(* CODESYS project DrugiiiiiZadatak (1).project
   CustomField04_name: CustomField04
   CustomField06_name: CustomField06
   CustomField07_name: CustomField07
   CustomField09_name: CustomField09
   CustomField08_name: CustomField08
   CustomField02_name: CustomField02
   CustomField10_name: CustomField10
   CustomField01_name: CustomField01
   CustomField03_name: CustomField03
   CustomField05_name: CustomField05

Project tree, tasks and I/O mapping:
  MyController : TM238LFDC24DT, Schneider Electric, order no. TM238LFDC24DT, version 2.0.31.8
    application Application
      task MAST (cyclic, interval 20 ms, priority 15, watchdog 100 ms x 1) calls POU
      function HiddenPOU [ST]
      global variables GVL
      program POU [LD]
    CAN
    Embedded Functions
      HSC : HSC, Schneider Electric, version 2.0.31.8
        HSC
      PTO_PWM : PTO_PWM, Schneider Electric, version 2.0.31.8
        PTO_PWM
      IO : IO, Schneider Electric, version 2.0.31.8
          input  Application.POU.Tipkalo2 : BOOL  // IW0.I9
          input  Application.POU.Tipkalo1 : BOOL  // IW0.I10
          output Application.POU.Zelena1 : BOOL  // QW0.Q4
          output Application.POU.Zuta1 : BOOL  // QW0.Q5
          output Application.POU.Crvena1 : BOOL  // QW0.Q6
          unmapped channels: IW0, QW0
    Serial Line 1
      Modbus_Manager : Modbus_Manager, Schneider Electric, version 2.0.1.12
    Serial Line 2
      SoMachine_Network_Manager : SoMachine-Network_Manager, Schneider Electric, version 2.0.1.10
  MachineLayoutPicture
*)

// MyController/Application/GVL
VAR_GLOBAL
END_VAR

// MyController/Application/POU
PROGRAM POU
VAR
	Tipkalo1: BOOL;
	Tipkalo2: BOOL;
	brojilo: CTUD := (CV := 5, RESET := FALSE, PV := 0, LOAD := FALSE, CD := FALSE, CU := FALSE, QD := FALSE, QU := FALSE);
	Zelena1: BOOL;
	Crvena1: BOOL;
	Zuta1: BOOL;
	
	
	titraj1: TP := (Q := TRUE, PT := TIME#5000ms, ET := TIME#5000ms, IN := TRUE);
	pomocni: TP := (Q := TRUE, PT := TIME#400MS, ET := TIME#400MS, IN := FALSE);
	pomocni1: TON := (Q := FALSE, PT := TIME#400ms, ET := TIME#0ms, IN := FALSE);
	pomocni3: TON := (Q := TRUE, PT := TIME#400MS, ET := TIME#0MS, IN := TRUE);
END_VAR

VAR_OUTPUT
	
END_VAR

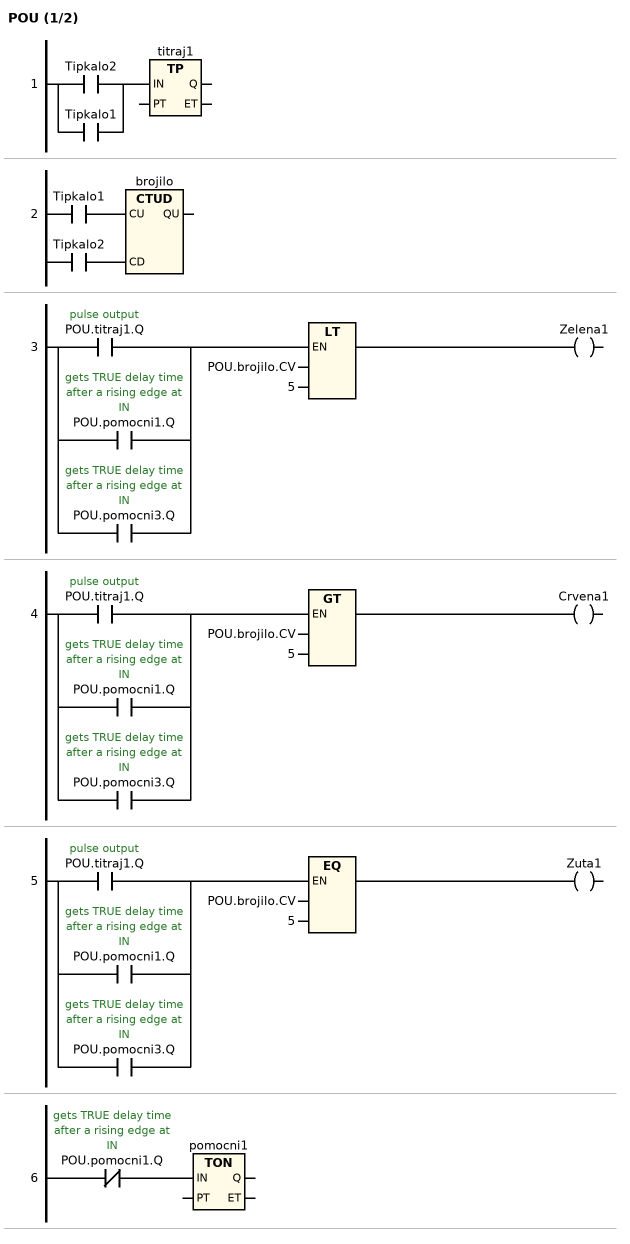
// NETWORK 1
titraj1(IN := Tipkalo2 OR Tipkalo1); // TP

// NETWORK 2
brojilo(CU := Tipkalo1, CD := Tipkalo2); // CTUD

// NETWORK 3
//   POU.titraj1.Q: pulse output
//   POU.pomocni1.Q: gets TRUE delay time after a rising edge at IN
//   POU.pomocni3.Q: gets TRUE delay time after a rising edge at IN
//   POU.brojilo.CV: Current Counter Value
Zelena1 := (POU.titraj1.Q OR POU.pomocni1.Q OR POU.pomocni3.Q) AND POU.brojilo.CV < 5;

// NETWORK 4
//   POU.titraj1.Q: pulse output
//   POU.pomocni1.Q: gets TRUE delay time after a rising edge at IN
//   POU.pomocni3.Q: gets TRUE delay time after a rising edge at IN
//   POU.brojilo.CV: Current Counter Value
Crvena1 := (POU.titraj1.Q OR POU.pomocni1.Q OR POU.pomocni3.Q) AND POU.brojilo.CV > 5;

// NETWORK 5
//   POU.titraj1.Q: pulse output
//   POU.pomocni1.Q: gets TRUE delay time after a rising edge at IN
//   POU.pomocni3.Q: gets TRUE delay time after a rising edge at IN
//   POU.brojilo.CV: Current Counter Value
Zuta1 := (POU.titraj1.Q OR POU.pomocni1.Q OR POU.pomocni3.Q) AND POU.brojilo.CV = 5;

// NETWORK 6
//   POU.pomocni1.Q: gets TRUE delay time after a rising edge at IN
pomocni1(IN := NOT POU.pomocni1.Q); // TON

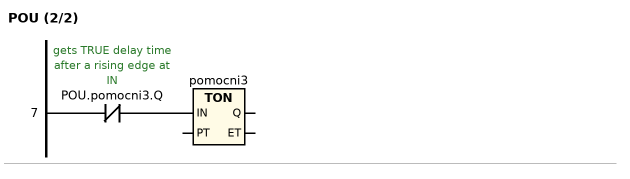
// NETWORK 7
//   POU.pomocni3.Q: gets TRUE delay time after a rising edge at IN
pomocni3(IN := NOT POU.pomocni3.Q); // TON

END_PROGRAM

// MyController/Application/HiddenPOU
FUNCTION HiddenPOU : BOOL

VAR_INPUT
	pHiddenFunc: POINTER TO WORD;
END_VAR
VAR
	pRead: POINTER TO BYTE;
	pWrite: POINTER TO BYTE;
END_VAR

pRead := pHiddenFunc + 400;
pWrite := pHiddenFunc + 4400;
HiddenPOU := TRUE;

END_FUNCTION
